// Struckig
// Copyright (C) 2022 Stefan Besler

// This program is free software: you can redistribute it and/or modify
// it under the terms of the GNU General Public License as published by
// the Free Software Foundation, either version 3 of the License, or
// (at your option) any later version.

// This program is distributed in the hope that it will be useful,
// but WITHOUT ANY WARRANTY; without even the implied warranty of
// MERCHANTABILITY or FITNESS FOR A PARTICULAR PURPOSE.  See the
// GNU General Public License for more details.
//
// You should have received a copy of the GNU General Public License
// along with THIS PROGRAM.  IF NOT, see <http://www.gnu.org/licenses/>.
{attribute 'qualified_only'}
/// Global configuration constants for Struckig.
/// These values define library limits and algorithm defaults that are
/// referenced by trajectory generation and numerical helper routines.
VAR_GLOBAL CONSTANT
  MaxDoFs : INT := 7; //< Maximum number of degrees of freedom supported by `Otg`.
  MaxIterations : BYTE := 127; //< Maximum iterations when [shrinking an interval](xref:Struckig.Roots#ShrinkInterval)
  NumericalRobust : BOOL := TRUE; //< Enables additional guards for numerically robust calculations.
  
  /// Default initial value for Otg.SmoothBrake / Otg1.SmoothBrake
  /// If enabled, braking profiles prefer smooth acceleration transitions.
  SmoothBrake : BOOL := FALSE;
END_VAR

(* stored: Version 1.1.0.1
   GVL ParameterList: Id {6cef246a-2041-4266-a931-0bae0d434120}, ParameterList True *)
